{attribute addProperty BoxType "EP9521-0020-0000"}
{attribute addProperty Id "A_0025_EP9576_1032_0016EP9576_B5DF83EF23229"}
{attribute addProperty CRC "1394071456"}
{attribute addProperty SizeInBites "232"}
{attribute addProperty SizeInBytes "29"}
TYPE A_0024_EP9521_0020_0000_5317D7A0 EXTENDS EP9521_179A0949 :
STRUCT
	{attribute addProperty Name "A_0025_EP9576_1032_0016"}
	A_0025_EP9576_1032_0016 : EP9576_B5DF83EF;
END_STRUCT
END_TYPE

(* stored: Version 1.2.0.0, ProductVersion 3.1.4024.9
   DUT A_0024_EP9521_0020_0000_5317D7A0: Id {c1f3d7ae-fca0-4cf9-a3a2-a4857f5815cb} *)
